FUNCTION_BLOCK XtsEnableSequence IMPLEMENTS ITask
VAR_INPUT
END_VAR
VAR_OUTPUT
END_VAR
VAR
	_collisionGroup : ICollisionGroup;
	addMover : AddMoverToGroupTask(_collisionGroup);
	moverNumbers : DINT;
	AllMoversEnabled: BOOL;
	EnableTrigger : BOOL;	
	Logger : TcMessage_Ext;
	State : INT;
	_busy : BOOL;
	_done : BOOL;
	_Error : BOOL;
END_VAR
VAR_IN_OUT
	arrMovers : ARRAY[*] OF IMover;
END_VAR

CASE State OF
	0:
		IF EnableTrigger THEN
			State := 10;
			EnableTrigger := FALSE;
			moverNumbers := 1;
			_busy := TRUE;
			_done := FALSE;
			_Error := FALSE;
		END_IF
		
	10:
		FOR moverNumbers := LOWER_BOUND(arrMovers,1) TO UPPER_BOUND(arrMovers,1) DO
			arrMovers[moverNumbers].ResetAxis();
		END_FOR
		moverNumbers := 1;
		State := 20;
		
	20:
		IF _collisionGroup.GroupState = CAGroupStatus.mcGroupStateErrorStop THEN
			_collisionGroup.Reset();
			Logger.Send(TC_EVENTS.XtsCAGroupEvents.CAGroupReset,'');
		END_IF
		State := 30;
		
	30:
		arrMovers[moverNumbers].IdentInGroup := DINT_TO_INT( moverNumbers);
		addMover.AddMover(MoverToAdd := arrMovers[moverNumbers]);
		logger.Send(TC_EVENTS.XtsCAGroupEvents.AddingMoverToGroup,DINT_TO_STRING(moverNumbers));
		State := 40;
		
	40:
		IF addMover.Done THEN
			IF moverNumbers <> UPPER_BOUND(arrMovers,1) THEN
				moverNumbers := moverNumbers + 1;
				State := 30;
			ELSE
				logger.Send(TC_EVENTS.XtsCAGroupEvents.AllMoversAdded,'');
				FOR moverNumbers := LOWER_BOUND(arrMovers,1) TO UPPER_BOUND(arrMovers,1) DO
					arrMovers[moverNumbers].EnableAxis();
				END_FOR
				State := 50;
			END_IF
		END_IF
		
	50:
		AllMoversEnabled := TRUE;
		FOR moverNumbers := LOWER_BOUND(arrMovers,1) TO UPPER_BOUND(arrMovers,1) DO
			AllMoversEnabled := TRUE AND arrMovers[moverNumbers].isEnabled();
		END_FOR
		IF AllMoversEnabled THEN
			logger.Send(TC_EVENTS.XtsCAGroupEvents.AllMoversEnabled,'');
			_collisionGroup.Enable();
			logger.Send(TC_EVENTS.XtsCAGroupEvents.CAGroupEnable,'');
			State := 60;
		END_IF
		
	60:
		IF _collisionGroup.GroupState = 2 THEN
			State := 0;
			_busy := FALSE;
			_done := true;
		END_IF
END_CASE

addMover();

METHOD Abort : BOOL
EnableTrigger := FALSE;
State := 0;
addMover.Abort();
END_METHOD

PROPERTY Busy : BOOL
GET
Busy := _busy;
END_GET
END_PROPERTY

PROPERTY Done : BOOL
GET
Done := _done;
END_GET
END_PROPERTY

METHOD Enable : BOOL
VAR_INPUT
END_VAR
IF NOT _busy THEN
	EnableTrigger := Enable := true;
END_IF
END_METHOD

PROPERTY Error : BOOL
GET
Error := _Error;
END_GET
END_PROPERTY

METHOD FB_init : BOOL
VAR_INPUT
	bInitRetains : BOOL; // if TRUE, the retain variables are initialized (warm start / cold start)
	bInCopyCode : BOOL;  // if TRUE, the instance afterwards gets moved into the copy code (online change)
	collisionGroup : ICollisionGroup;
END_VAR
_collisionGroup := collisionGroup;
addMover.FB_init(FALSE, FALSE, collisionGroup);
END_METHOD

END_FUNCTION_BLOCK

(* stored: Version 1.1.0.1, ProductVersion 3.1.4024.12
   POU XtsEnableSequence: Id {b3bae6c3-ef72-4837-b4e0-3c1e6cb08595}, SpecialFunc None
   Method Abort: Id {cafb98cb-e0e4-409c-b6f8-122c787fc07d}
   Property Busy: Id {46653790-8548-49c2-8cf9-461f616a7413}
   Get Get: Id {2914fa43-f085-4d43-9500-5b40f3cbed00}
   Property Done: Id {3d3bebc9-a410-4875-8a42-cd9e32cd3fab}
   Get Get: Id {37ccb39e-1d6a-4c57-8922-2c7d24188f37}
   Method Enable: Id {1d42943b-c792-49a8-a140-4271fe755723}
   Property Error: Id {301d19ed-98b9-48e7-887b-89163b0ce3ad}
   Get Get: Id {4cbf8de7-2404-46d3-8c55-b82ac3a79fd9}
   Method FB_init: Id {a774c049-4849-459f-b124-c9b64376f790} *)
